{attribute 'pack_mode' := '1'} 
TYPE MYSTRUCT :
STRUCT
	a : BOOL;
	b : INT;
	c : DINT;
END_STRUCT
END_TYPE

(* stored: Version 1.1.0.1, ProductVersion 3.1.4024.11
   DUT MYSTRUCT: Id {292a9d60-527d-4dac-9e6e-0220928ad7a5} *)
